# EPICS substitutions: ek9000App/Db/EL1001.substitutions
file EL1001.template
{ 	pattern
	{
		TERMINAL,
		DESC1,	ZNAM1,	ONAM1,	ZSV1,	OSV1,	COSV1,	SCAN1
	}
	{
	}
}
